(* IEC 61131-3 sources: volt/packages/volt-lsp-iec/test-corpus/pro2193/Device/Plc Logic/Application/09 Misc/Library Manager/(unresolved)/collections interfaces, 5 files *)

(* ---- INSTANCEPATHBUILDINGNODETYPE.dut ---- *)
TYPE INSTANCEPATHBUILDINGNODETYPE :
(
	STRUCTUREDNODE,
	ARRAYNODE,
	POINTERNODE,
	VALUENODE
);
END_TYPE

(* ---- INTERFACEIDS.gvl ---- *)
VAR_GLOBAL
	ITFID_IBASETREENODE : DWORD := 16#1003;
	ITFID_INAMEDTREENODE : DWORD := 16#1004;
	ITFID_IINSTANCEPATHBUILDINGNODE : DWORD := 16#1005;
END_VAR

(* ---- IBASETREENODE.itf ---- *)
INTERFACE IBASETREENODE
END_INTERFACE

METHOD GETCHILD : IBaseTreeNode
VAR_INPUT
	DIINDEX : DINT;
END_VAR
END_METHOD

METHOD GETFATHER : IBaseTreeNode
END_METHOD

(* ---- IINSTANCEPATHBUILDINGNODE.itf ---- *)
INTERFACE IINSTANCEPATHBUILDINGNODE
END_INTERFACE

METHOD GETFULLPATH : DINT
VAR_INPUT
	PBUFFER : POINTER TO STRING;
	DIBUFFERSIZE : DINT;
END_VAR
END_METHOD

METHOD PRVDOGETFULLPATH : DINT
VAR_INPUT
	PBUFFER : POINTER TO STRING;
	DIBUFFERSIZE : DINT;
END_VAR
END_METHOD

(* ---- INAMEDTREENODE.itf ---- *)
INTERFACE INAMEDTREENODE
END_INTERFACE

METHOD ABSTRCOMPARETO : INT
VAR_INPUT
	PSEARCHDATA : POINTER TO BYTE;
END_VAR
END_METHOD

METHOD FINDCHILDBYNAME : INamedTreeNode
VAR_INPUT
	STNAME : STRING(256);
END_VAR
END_METHOD
